Staubli VAL3: CircleCenter.dtx

bool bExit
public bool bFrameSave
bool bFrameTeach = true
bool bOk = true
bool bSame = true
frame fFrame1 = {x=1609.698381, y=34.606682, z=-207.653176, rx=4.827804, ry=-0.339181, rz=5.164815, fatherId=world[0]}
frame fFrameRef = {fatherId=world[0]}
mdesc mNomSpeed
num nAngle = 7.0664356
num nDia = 264.172018
num nFrame1Err
num nItem[6]
num nMax[6]
num nMin[6]
num nSelectedPt = 2
num nStatus = 6
num nWorkingMode = 1
public pointRx pFrameRefPt[3]
  [0] = {x=1741.245798, y=46.389469, z=-205.876469, rx=0.131165, ry=-179.946881, rz=21.208274, shoulder=lefty, elbow=epositive, wrist=wpositive, fatherId=world[0]}
  [1] = {x=1608.405084, y=166.218402, z=-196.544793, rx=0.131429, ry=-179.945224, rz=21.207967, shoulder=lefty, elbow=epositive, wrist=wpositive, fatherId=world[0]}
  [2] = {x=1609.086584, y=-73.34702, z=-195.821119, rx=0.131457, ry=-179.944094, rz=21.208415, shoulder=lefty, elbow=epositive, wrist=wpositive, fatherId=world[0]}
pointRx pPointCenter = {x=1609.698381, y=34.606682, z=-207.653176, rx=4.827804, ry=-0.339181, rz=137.862918, fatherId=world[0]}
string sButton[2]
  [0] = "是"
  [1] = "否"
string sCutPosStatus
string sEmptyOrNotC[3]
string sItem[6]
string sOffSet[6]
  [0] = "X:  1609.7 "
  [1] = "Y:  34.61"
  [2] = "Z:  -207.65"
  [3] = "Rx: 4.83"
  [4] = "Ry: -0.34"
  [5] = "Rz: 5.16"
string sThreeOffset[3]
  [0] = "第1点(圆周上)"
  [1] = "第2点(圆周上)"
  [2] = "第3点(圆周上)"
tool tTool = {x=350.22, y=-0.767094, z=232.538993, rx=-89.841339, ry=89.729222, rz=89.842087, fatherId=flange[0], ioLink=valve1}
trsf trFrame
trsf trOffSetOut
trsf trOffset = {x=1609.698381, y=34.606682, z=-207.653176, rx=4.827804, ry=-0.339181, rz=5.164815}
